// TIA Portal V16 export
// export: Created 2023-03-29T11:04:57.8810626Z, ExportSetting WithDefaults, DisplayName Totally Integrated Automation Portal, DisplayVersion V16 Update 6, DisplayName TIA Portal Version Control Interface, DisplayVersion V16 Update 2, DisplayName TIA Portal Openness, DisplayVersion V16 Update 6, DisplayName STEP 7 Professional, DisplayVersion V16 Update 6, DisplayName STEP 7 Safety, DisplayVersion V16, DisplayName WinCC Advanced, DisplayVersion V16 Update 6
DATA_BLOCK "dbControl of compressor conection network"   // DB47
AUTHOR : rtecmer
VERSION : 0.1
// stored: AutoNumber true, DBAccessibleFromOPCUA true, InstanceOfName Sterowanie dołączeniem na sieć, InstanceOfType FB
"Sterowanie dołączeniem na sieć"
   // VAR_INPUT
   //    IsReady_M : Bool;
   //    IsModeAut : Bool;
   //    Time_Off_Inverter : Bool;
   //    setMotor2 : Bool;
   //    setMotor3 : Bool;
   //    setMotor4 : Bool;
   //    IsRunNetwork_M : Bool;
   //    CMD_A_NetworkM : Bool;
   // END_VAR
   // VAR_IN_OUT
   //    TimerStartNetworkContactor : TON_TIME;
   //    setCMD_SM : Bool;
   //    Is_extras_K1_M_1 : Bool;
   //    Is_extras_K2_M_1 : Bool;
   //    Is_extras_K3_M_1 : Bool;
   //    setSUPV_SM : Bool;
   //    off_add_K1 : Bool;
   //    off_add_K2 : Bool;
   //    off_add_K3 : Bool;
   // END_VAR
BEGIN
END_DATA_BLOCK
